// TIA Portal V18 export
VAR_GLOBAL   // PLC tag table "Cabinet_9"
   Sz9_Button_LED_ST09_ST10 AT %Q1900.0 : Bool;
   Sz9_Button_LED_ST10_ST11 AT %Q1900.1 : Bool;
   Sz9_ST09_SenA AT %I1900.0 : Bool;
   Sz9_ST09_SenB AT %I1900.1 : Bool;
   Sz9_ST09_SenC AT %I1900.2 : Bool;
   Sz9_ST09_SenD AT %I1900.3 : Bool;
   Sz9_ST10_SenA AT %I1900.4 : Bool;
   Sz9_ST10_SenB AT %I1900.5 : Bool;
   Sz9_ST10_SenC AT %I1900.6 : Bool;
   Sz9_ST10_SenD AT %I1900.7 : Bool;
   Sz9_Button_ST09_ST10 AT %I1901.0 : Bool;
   Sz9_Button_ST10_ST11 AT %I1901.1 : Bool;
   "Reserved(126)" AT %I1901.2 : Bool;
   "Reserved(127)" AT %I1901.3 : Bool;
   "Reserved(128)" AT %I1901.4 : Bool;
   "Reserved(129)" AT %I1901.5 : Bool;
   "Reserved(130)" AT %I1901.6 : Bool;
   "Reserved(131)" AT %I1901.7 : Bool;
   Sz9_Safety1_1 AT %I1950.0 : Bool;
   Sz9_Safety1_2 AT %I1950.4 : Bool;
   "Reserved(132)" AT %I1950.1 : Bool;
   "Reserved(133)" AT %I1950.2 : Bool;
   "Reserved(134)" AT %I1950.3 : Bool;
   "Reserved(135)" AT %I1950.5 : Bool;
   "Reserved(136)" AT %I1950.6 : Bool;
   "Reserved(137)" AT %I1950.7 : Bool;
   "Reserved(138)" AT %I1951.0 : Bool;
   "Reserved(139)" AT %I1951.1 : Bool;
   "Reserved(140)" AT %I1951.2 : Bool;
   "Reserved(141)" AT %I1951.3 : Bool;
   "Reserved(142)" AT %I1951.4 : Bool;
   "Reserved(143)" AT %I1951.5 : Bool;
   "Reserved(144)" AT %I1951.6 : Bool;
   "Reserved(145)" AT %I1951.7 : Bool;
END_VAR
